PROGRAM InductiveSensor
VAR
	fbSensor	: FB_Component_InductiveSensor;
END_VAR

fbSensor(	sName		:= 'Inductive Sensor Test',
			bEnable		:= TRUE,
			bRawSignal	:= GVL.bWire1NotAvailable,
			tDebounce	:= T#0MS,
			tTimeOut	:= T#0MS);

END_PROGRAM

(* stored: Version 1.1.0.1, ProductVersion 3.1.4024.15
   POU InductiveSensor: Id {6d1e6f37-d7e9-4248-922e-a0fd41b35608}, SpecialFunc None *)
